FUNCTION_BLOCK WaterHeaterPlantODE (* ODE_fb *)
  (* Standard: 61499-2 *)
  (* Version 0.1, 2017-00-25, hpea485, UOA *)
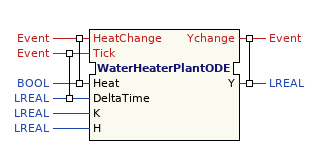
  EVENT_INPUT
    HeatChange WITH Heat;
    Tick WITH DeltaTime;
  END_EVENT
  EVENT_OUTPUT
    Ychange WITH Y;
  END_EVENT
  VAR_INPUT
    Heat : BOOL;
    DeltaTime : LREAL;
    K : LREAL;
    H : LREAL;
  END_VAR
  VAR_OUTPUT
    Y : LREAL;
  END_VAR
  VAR
    X : LREAL;
  END_VAR
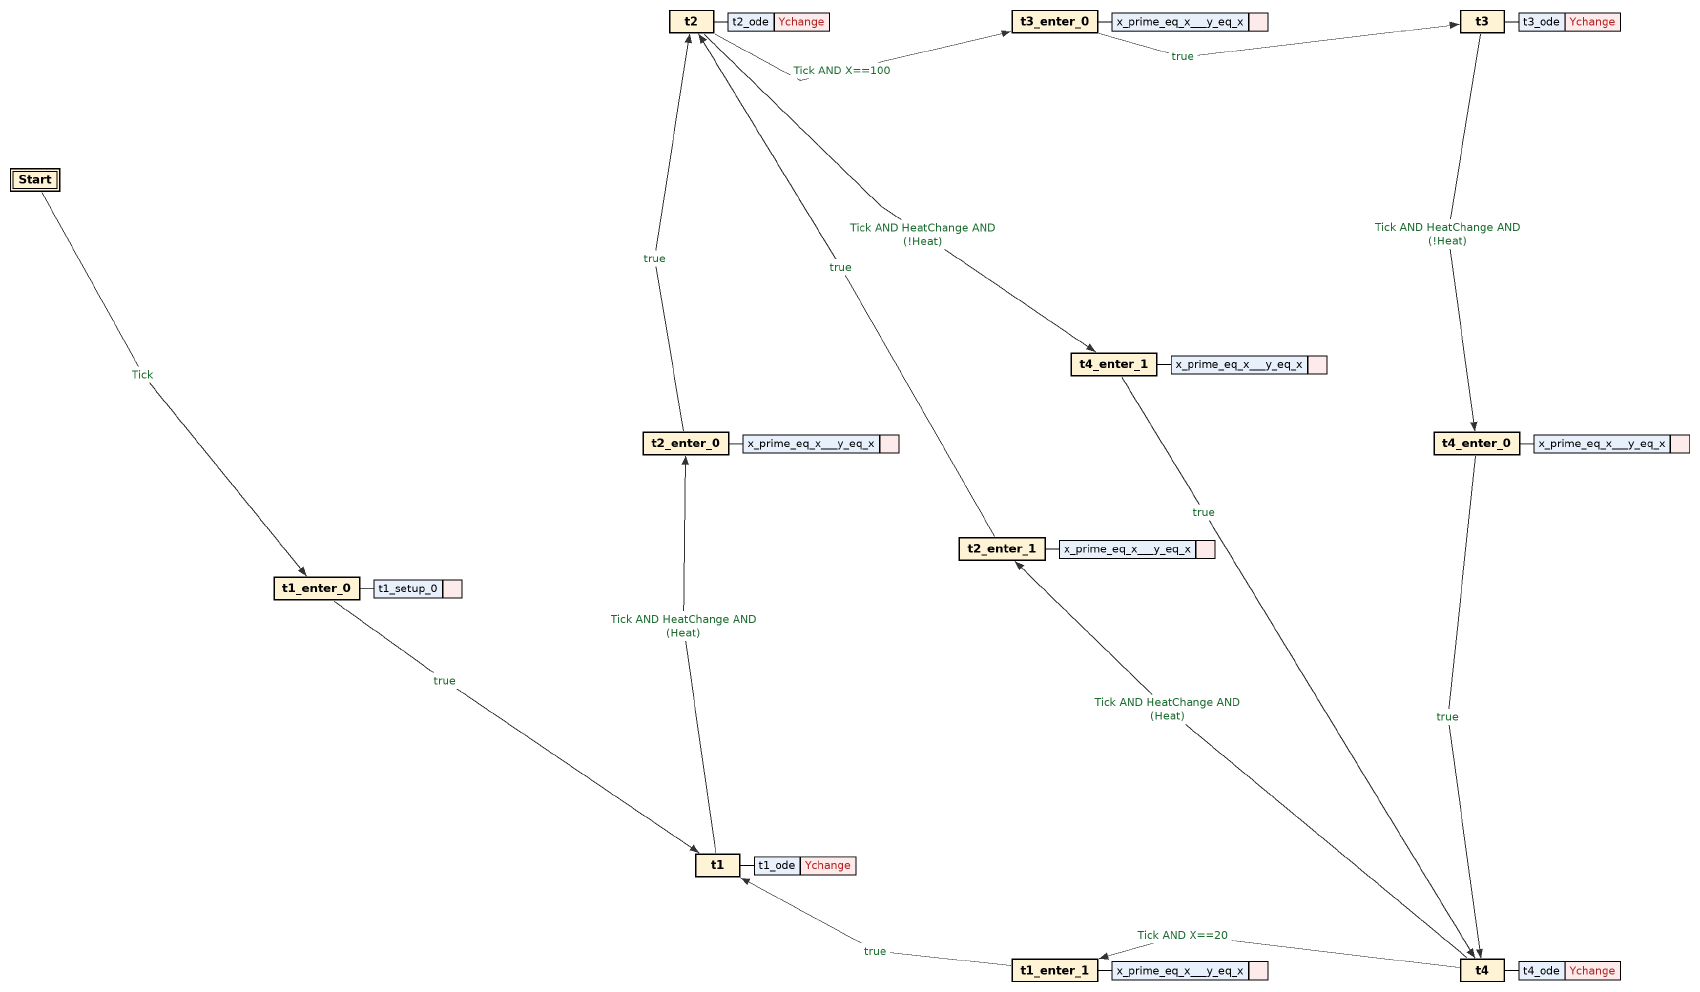
  EC_STATES
    Start;
    t1_enter_0 : t1_setup_0;
    t1 : t1_ode -> Ychange;
    t2_enter_0 : x_prime_eq_x___y_eq_x;
    t2 : t2_ode -> Ychange;
    t1_enter_1 : x_prime_eq_x___y_eq_x;
    t4 : t4_ode -> Ychange;
    t3_enter_0 : x_prime_eq_x___y_eq_x;
    t3 : t3_ode -> Ychange;
    t4_enter_0 : x_prime_eq_x___y_eq_x;
    t2_enter_1 : x_prime_eq_x___y_eq_x;
    t4_enter_1 : x_prime_eq_x___y_eq_x;
  END_STATES
  EC_TRANSITIONS
    Start TO t1_enter_0 := Tick;
    t1_enter_0 TO t1 := true;
    t1 TO t2_enter_0 := Tick AND HeatChange AND (Heat);
    t2_enter_0 TO t2 := true;
    t2 TO t3_enter_0 := Tick AND X==100;
    t2 TO t4_enter_1 := Tick AND HeatChange AND (!Heat);
    t1_enter_1 TO t1 := true;
    t4 TO t1_enter_1 := Tick AND X==20;
    t4 TO t2_enter_1 := Tick AND HeatChange AND (Heat);
    t3_enter_0 TO t3 := true;
    t3 TO t4_enter_0 := Tick AND HeatChange AND (!Heat);
    t4_enter_0 TO t4 := true;
    t2_enter_1 TO t2 := true;
    t4_enter_1 TO t4 := true;
  END_TRANSITIONS
  ALGORITHM t1_ode IN C: (* ODE *)
X_dot = 0;
Y = X;
  END_ALGORITHM
  ALGORITHM t1_setup_0 IN C: (* ODE_init *)
X_prime = 20;
Y = 20;
  END_ALGORITHM
  ALGORITHM t2_ode IN C: (* ODE *)
X_dot = K * (H - X);
Y = X;
X_trigger = 100;
  END_ALGORITHM
  ALGORITHM x_prime_eq_x___y_eq_x IN C: (* ODE_init *)
X_prime = X;
Y = X;
  END_ALGORITHM
  ALGORITHM t3_ode IN C: (* ODE *)
X_dot = 0;
Y = X;
  END_ALGORITHM
  ALGORITHM t4_ode IN C: (* ODE *)
X_dot = -K * X;
Y = X;
X_trigger = 20;
  END_ALGORITHM
END_FUNCTION_BLOCK
